FUNCTION_BLOCK ScaleFB
VAR_INPUT
	iRohWert: INT;
END_VAR
VAR_OUTPUT
	ScaledValue: INT;
END_VAR
VAR
	NormMIN:INT:= 0;
	NormMAX:INT:= 27648;
	ScaleMIN:INT:= 0;
	ScaleMAX:INT:= 100;
END_VAR

ScaledValue:= ((ScaleMAX-ScaleMIN)*(iRohWert-NormMIN)/(NormMAX-NormMIN))+ScaleMIN;

END_FUNCTION_BLOCK

(* stored: Version 1.1.0.1
   POU ScaleFB: Id {d354267a-1e40-491c-97cd-56fb94a43883}, SpecialFunc None *)
